{attribute 'linkalways'}
{attribute 'hide_all_locals'}
FUNCTION_BLOCK ValueString EXTENDS ValueStringRead IMPLEMENTS Value
VAR
END_VAR

METHOD SetFromType : BOOL
VAR_INPUT
	source : __SYSTEM.AnyType;
END_VAR
SetFromType := ConvertAnyType(source, thisAnyType);
END_METHOD

METHOD SetFromString : BOOL
VAR_INPUT
	value : T_MaxString;
END_VAR
thisValue := value;

SetFromString := TRUE;
END_METHOD

METHOD Set : BOOL
VAR_INPUT
	source : ANY;
END_VAR
Set := ConvertAnyType(source, thisAnyType);
END_METHOD

END_FUNCTION_BLOCK

(* stored: Version 1.1.0.1
   POU ValueString: Id {ef85f8f4-0525-4520-8875-5621a15fb963}, SpecialFunc None
   Method SetFromType: Id {7ef82213-81ac-4b7b-aea2-5eb477c9dcea}
   Method SetFromString: Id {3ae95eac-0357-4065-8311-55b9de4b7b98}
   Method Set: Id {069cfadf-e251-47dc-84ec-611b44a31cbe} *)
